Fanuc KAREL source: NC0009.KL

-- PROVISIONAL review KL for V940-1; original PC SHA256 3af8d6bfef298f3560eb4380ad5ade8922ff813a3085d8efcac00fb756596cdb
-- Incomplete behavior may be omitted. Consult companion uncertainty JSON. Do not deploy.
PROGRAM NC0009
%NOLOCKGROUP
-- UNRESOLVED_LOCAL_POOL 1 cells at code offset 3; source declarations unknown
-- DIRECT_LOCAL_WORD_ACCESS alone does not prove INTEGER, REAL, or BOOLEAN
BEGIN
  -- V9_EXPOSED_INDEXED_TABLE_HINT layout=0001; 30 counted words exposed once; source arms/runtime held
  -- V9_CONDITION_STACK_HINT 15 bounded expression windows; static native code-base-relative target link; source arms held
  -- UNRESOLVED_PC offsets 0-8; opcodes 2B,2C,7B
  -- UNRESOLVED_PC offsets 13-20; opcodes 9D,23
  -- UNRESOLVED_PC offsets 25-38; opcodes 21,9D,57,79
  -- UNRESOLVED_PC offsets 43-56; opcodes 21,9D,57,79
  -- UNRESOLVED_PC offsets 61-74; opcodes 21,9D,57,79
  -- UNRESOLVED_PC offsets 79-92; opcodes 21,9D,57,79
  -- UNRESOLVED_PC offsets 97-110; opcodes 21,9D,57,79
  -- UNRESOLVED_PC offsets 115-128; opcodes 21,9D,57,79
  -- UNRESOLVED_PC offsets 133-146; opcodes 21,9D,57,79
  -- UNRESOLVED_PC offsets 151-164; opcodes 21,9D,57,79
  -- UNRESOLVED_PC offsets 169-182; opcodes 21,9D,57,79
  -- UNRESOLVED_PC offsets 187-200; opcodes 21,9D,57,79
  -- UNRESOLVED_PC offsets 205-218; opcodes 21,9D,57,79
  -- UNRESOLVED_PC offsets 223-236; opcodes 21,9D,57,79
  -- UNRESOLVED_PC offsets 241-254; opcodes 21,9D,57,79
  -- UNRESOLVED_PC offsets 259-272; opcodes 21,9D,57,79
  -- UNRESOLVED_PC offsets 277-290; opcodes 21,9D,57,79
  -- UNRESOLVED_PC offsets 295-309; opcodes 21,9D,52,23
  -- UNRESOLVED_PC offsets 314-319; opcodes 7A
  -- UNRESOLVED_PC offsets 324-342; opcodes 21,2E,52,23
  -- UNRESOLVED_PC offsets 352-357; opcodes 7A
  -- UNRESOLVED_PC offsets 362-380; opcodes 21,2E,52,23
  -- UNRESOLVED_PC offsets 390-395; opcodes 7A
  -- UNRESOLVED_PC offsets 400-418; opcodes 21,2E,52,23
  -- UNRESOLVED_PC offsets 428-433; opcodes 7A
  -- UNRESOLVED_PC offsets 438-456; opcodes 21,2E,52,23
  -- UNRESOLVED_PC offsets 466-471; opcodes 7A
  -- UNRESOLVED_PC offsets 476-494; opcodes 21,2E,52,23
  -- UNRESOLVED_PC offsets 504-509; opcodes 7A
  -- UNRESOLVED_PC offsets 514-532; opcodes 21,2E,52,23
  -- UNRESOLVED_PC offsets 542-547; opcodes 7A
  -- UNRESOLVED_PC offsets 552-570; opcodes 21,2E,52,23
  -- UNRESOLVED_PC offsets 580-585; opcodes 7A
  -- UNRESOLVED_PC offsets 590-608; opcodes 21,2E,52,23
  -- UNRESOLVED_PC offsets 618-623; opcodes 7A
  -- UNRESOLVED_PC offsets 628-646; opcodes 21,2E,52,23
  -- UNRESOLVED_PC offsets 656-661; opcodes 7A
  -- UNRESOLVED_PC offsets 666-684; opcodes 21,2E,52,23
  -- UNRESOLVED_PC offsets 694-699; opcodes 7A
  -- UNRESOLVED_PC offsets 704-722; opcodes 21,2E,52,23
  -- UNRESOLVED_PC offsets 732-737; opcodes 7A
  -- UNRESOLVED_PC offsets 742-760; opcodes 21,2E,52,23
  -- UNRESOLVED_PC offsets 770-775; opcodes 7A
  -- UNRESOLVED_PC offsets 780-798; opcodes 21,2E,52,23
  -- UNRESOLVED_PC offsets 808-813; opcodes 7A
  -- UNRESOLVED_PC offsets 818-836; opcodes 21,2E,52,23
  -- UNRESOLVED_PC offsets 846-851; opcodes 7A
  -- UNRESOLVED_PC offsets 856-874; opcodes 21,2E,52,23
  -- UNRESOLVED_PC offsets 884-888; opcodes 7F
  -- UNRESOLVED_PC offsets 893-897; opcodes 27,AA
  -- UNRESOLVED_PC offsets 902-906; opcodes 7F
END NC0009
